Staubli VAL3: resetAllPallet.pgx

program resetAllPallet()
  local num i
  local string l_sPalletName
begin
  // resetALL
  call pallet:reset()
  // call the onEvent procedure
  call OnEvent:OnCycleEvent(16)
end
